# EPICS substitutions: db/Beckhoff_2XXX/ecmcEL2008.substitutions
file "ecmcEcSlave.template"
{
  pattern {}
          {}
}

file "ecmc_binaryOutput-chX.template"
{
  pattern {CH_ID}
          {01   }
          {02   }
          {03   }
          {04   }
          {05   }
          {06   }
          {07   }
          {08   }
}
